PROGRAM Step_6_Log_Sequence
VAR
	j, i: INT;
	
	SelectedFoot   : INT := 0;   // 0 = none, otherwise 4..16
    //GVL ---------ConfirmedFoot  : INT := 0;   // Confirmed length
    rtConfirm      : R_TRIG;     // for one-shot on ConfirmPB
	rtCancel : R_TRIG;   // edge detector for Cancel
END_VAR





// One-shot on Confirm button
rtConfirm(CLK := ConfirmPB);
// One-shot on Cancel button
rtCancel(CLK := CancelPB);







// If a PB is pressed, set that light ON and others OFF
FOR j := 4 TO 16 DO
    IF PBFoot[j] THEN
        // turn all lights off first
        FOR i := 4 TO 16 DO
            LTFoot[i] := FALSE;
        END_FOR;
		
        // turn only this one ON
        LTFoot[j] := TRUE;
		
		// remember which length is selected
        SelectedFoot := j;   // j will be 4..16
    END_IF;
END_FOR;

//-------------------------------------------------------------------------------------

// One-shot on Confirm button
IF rtConfirm.Q THEN
    // Save the current selected length
    ConfirmedFoot := SelectedFoot;

    // Add it into the FIFO (first empty slot)
    FOR i := 1 TO 5 DO
        IF FootFIFO[i] = 0 THEN
            FootFIFO[i] := ConfirmedFoot;   // store new graded length
            EXIT;                           // stop after writing one slot
        END_IF;
    END_FOR;

    // 3) Clear the lights and selection ready for next board
    FOR j := 4 TO 16 DO
        LTFoot[j] := FALSE;
    END_FOR;

    SelectedFoot := 0;
END_IF;
	
//-----------------------------------------------------------------------------------
// One-shot on Cancel button
IF rtCancel.Q THEN
    // Remove the newest board entered by the grader.
    //  start from the back (slot 5) and clear the first non-zero we find.
    FOR i := 5 TO 1 BY -1 DO
        IF FootFIFO[i] <> 0 THEN // <> "Not equal to"
            FootFIFO[i] := 0;          // clear that newest entry
            EXIT;                      // stop after clearing one
        END_IF;
    END_FOR;
END_IF;

END_PROGRAM

(* stored: Version 1.1.0.1
   POU Step_6_Log_Sequence: Id {3303b1f5-236e-4467-934a-57e2043a7a2d}, SpecialFunc None *)
